// TIA Portal V17 export
// export: Created 2026-08-04T13:53:45.7641817Z, ExportSetting WithDefaults, DisplayName Totally Integrated Automation Portal, DisplayVersion V17, DisplayName TIA Portal Openness, DisplayVersion V17, DisplayName TIA Portal Version Control Interface, DisplayVersion V17, DisplayName SINAMICS Startdrive Advanced, DisplayVersion V17, DisplayName SINAMICS Startdrive G130, G150, S120, S150, SINAMICS MV, G220, S200, S210, DisplayVersion V17, DisplayName SINAMICS Startdrive G110M, G120, G120C, G120D, G120P, G115D, DisplayVersion V17, DisplayName STEP 7 Professional, DisplayVersion V17, DisplayName STEP 7 Safety, DisplayVersion V17, DisplayName WinCC Basic/Comfort/Advanced, DisplayVersion V17, DisplayName WinCC Unified, DisplayVersion V17
FUNCTION_BLOCK "Faults_FB"   // FB2, LAD
TITLE = Fault Detection
{ S7_Optimized_Access := 'TRUE' }
VERSION : 0.1
// Monitors process conditions and sets fault bits in Faults_UDT. Handles EStop detection, temperature faults, sensor health, switch conflicts, and active fault counting.
// stored: AutoNumber true, IsIECCheckEnabled false, IsRetainMemResEnabled false, MemoryReserve 100, SetENOAutomatically false, UDAEnableTagReadback false
   VAR
      Clear_Faults : "Faults_UDT";
      ons1 : Bool;
      highlimit : Real;
      TON : Array[0..10] of IEC_TIMER;
   END_VAR
   VAR_TEMP
      lowlimit : Real;
      faultcount : Int;
   END_VAR
   VAR_TEMP   // added for the SCL form of the ladder/FBD networks
      _w1 : Bool;
      _w2 : Bool;
   END_VAR
BEGIN

REGION Network 1: Fault Reset
   // Here we move a blank set of faults into our current active faults to reset them.
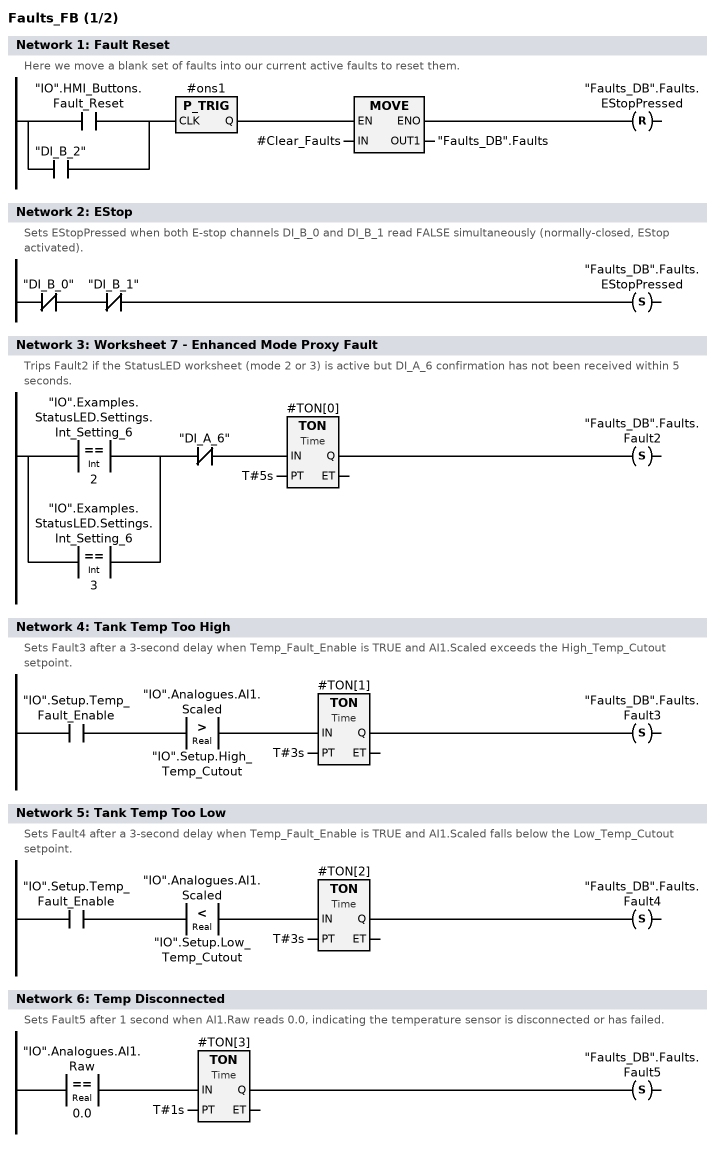
   RUNG wire#powerrail
      Contact( "IO".HMI_Buttons.Fault_Reset )
      wire#w1
      P_Trig( #ons1 )
      Move(in := #Clear_Faults, out1 => "Faults_DB".Faults)
      R_Coil( "Faults_DB".Faults.EStopPressed )
   END_RUNG
   RUNG wire#powerrail
      Contact( "DI_B_2" )
   END_RUNG wire#w1
   // the same network as SCL:
   #_w1 := "IO".HMI_Buttons.Fault_Reset OR "DI_B_2";
   #_w2 := #_w1 AND NOT #ons1;   // rising edge
   #ons1 := #_w1;
   IF #_w2 THEN
       "Faults_DB".Faults := #Clear_Faults;
       "Faults_DB".Faults.EStopPressed := FALSE;
   END_IF;
END_REGION

REGION Network 2: EStop
   // Sets EStopPressed when both E-stop channels DI_B_0 and DI_B_1 read FALSE simultaneously (normally-closed, EStop activated).
   RUNG wire#powerrail
      I_Contact( "DI_B_0" )
      I_Contact( "DI_B_1" )
      S_Coil( "Faults_DB".Faults.EStopPressed )
   END_RUNG
   // the same network as SCL:
   IF NOT "DI_B_0" AND NOT "DI_B_1" THEN "Faults_DB".Faults.EStopPressed := TRUE; END_IF;
END_REGION

REGION Network 3: Worksheet 7 - Enhanced Mode Proxy Fault
   // Trips Fault2 if the StatusLED worksheet (mode 2 or 3) is active but DI_A_6 confirmation has not been received within 5 seconds.
   RUNG wire#powerrail
      { S7_Templates := "SrcType := Int" } EQ_Contact(in1 := "IO".Examples.StatusLED.Settings.Int_Setting_6, in2 := 2)
      wire#w1
      I_Contact( "DI_A_6" )
      { S7_Templates := "time_type := Time" } #TON[0].TON(pt := T#5s, et =>)
      S_Coil( "Faults_DB".Faults.Fault2 )
   END_RUNG
   RUNG wire#powerrail
      { S7_Templates := "SrcType := Int" } EQ_Contact(in1 := "IO".Examples.StatusLED.Settings.Int_Setting_6, in2 := 3)
   END_RUNG wire#w1
   // the same network as SCL:
   #TON[0].TON(IN := (("IO".Examples.StatusLED.Settings.Int_Setting_6 = 2) OR ("IO".Examples.StatusLED.Settings.Int_Setting_6 = 3)) AND NOT "DI_A_6",
               PT := T#5s);
   IF #TON[0].Q THEN "Faults_DB".Faults.Fault2 := TRUE; END_IF;
END_REGION

REGION Network 4: Tank Temp Too High
   // Sets Fault3 after a 3-second delay when Temp_Fault_Enable is TRUE and AI1.Scaled exceeds the High_Temp_Cutout setpoint.
   RUNG wire#powerrail
      Contact( "IO".Setup.Temp_Fault_Enable )
      { S7_Templates := "SrcType := Real" } GT_Contact(in1 := "IO".Analogues.AI1.Scaled, in2 := "IO".Setup.High_Temp_Cutout)
      { S7_Templates := "time_type := Time" } #TON[1].TON(pt := T#3s, et =>)
      S_Coil( "Faults_DB".Faults.Fault3 )
   END_RUNG
   // the same network as SCL:
   #TON[1].TON(IN := "IO".Setup.Temp_Fault_Enable AND ("IO".Analogues.AI1.Scaled > "IO".Setup.High_Temp_Cutout),
               PT := T#3s);
   IF #TON[1].Q THEN "Faults_DB".Faults.Fault3 := TRUE; END_IF;
END_REGION

REGION Network 5: Tank Temp Too Low
   // Sets Fault4 after a 3-second delay when Temp_Fault_Enable is TRUE and AI1.Scaled falls below the Low_Temp_Cutout setpoint.
   RUNG wire#powerrail
      Contact( "IO".Setup.Temp_Fault_Enable )
      { S7_Templates := "SrcType := Real" } LT_Contact(in1 := "IO".Analogues.AI1.Scaled, in2 := "IO".Setup.Low_Temp_Cutout)
      { S7_Templates := "time_type := Time" } #TON[2].TON(pt := T#3s, et =>)
      S_Coil( "Faults_DB".Faults.Fault4 )
   END_RUNG
   // the same network as SCL:
   #TON[2].TON(IN := "IO".Setup.Temp_Fault_Enable AND ("IO".Analogues.AI1.Scaled < "IO".Setup.Low_Temp_Cutout),
               PT := T#3s);
   IF #TON[2].Q THEN "Faults_DB".Faults.Fault4 := TRUE; END_IF;
END_REGION

REGION Network 6: Temp Disconnected
   // Sets Fault5 after 1 second when AI1.Raw reads 0.0, indicating the temperature sensor is disconnected or has failed.
   RUNG wire#powerrail
      { S7_Templates := "SrcType := Real" } EQ_Contact(in1 := "IO".Analogues.AI1.Raw, in2 := 0.0)
      { S7_Templates := "time_type := Time" } #TON[3].TON(pt := T#1s, et =>)
      S_Coil( "Faults_DB".Faults.Fault5 )
   END_RUNG
   // the same network as SCL:
   #TON[3].TON(IN := "IO".Analogues.AI1.Raw = 0.0, PT := T#1s);
   IF #TON[3].Q THEN "Faults_DB".Faults.Fault5 := TRUE; END_IF;
END_REGION

REGION Network 7: AI0 Out of Bounds
   // Sets Fault6 after 1 second when AI0.Raw is outside the valid 0-28000 range, indicating a potentiometer fault or wiring issue.
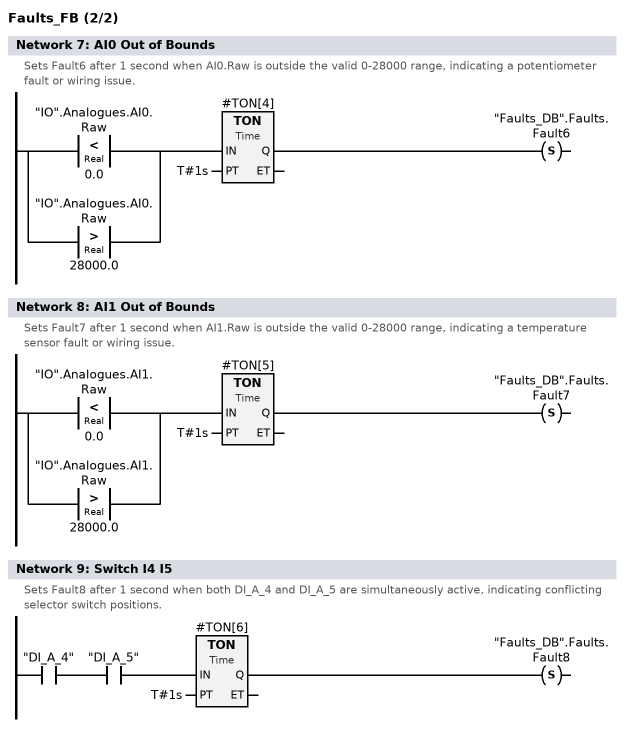
   RUNG wire#powerrail
      { S7_Templates := "SrcType := Real" } LT_Contact(in1 := "IO".Analogues.AI0.Raw, in2 := 0.0)
      wire#w1
      { S7_Templates := "time_type := Time" } #TON[4].TON(pt := T#1s, et =>)
      S_Coil( "Faults_DB".Faults.Fault6 )
   END_RUNG
   RUNG wire#powerrail
      { S7_Templates := "SrcType := Real" } GT_Contact(in1 := "IO".Analogues.AI0.Raw, in2 := 28000.0)
   END_RUNG wire#w1
   // the same network as SCL:
   #TON[4].TON(IN := ("IO".Analogues.AI0.Raw < 0.0) OR ("IO".Analogues.AI0.Raw > 28000.0), PT := T#1s);
   IF #TON[4].Q THEN "Faults_DB".Faults.Fault6 := TRUE; END_IF;
END_REGION

REGION Network 8: AI1 Out of Bounds
   // Sets Fault7 after 1 second when AI1.Raw is outside the valid 0-28000 range, indicating a temperature sensor fault or wiring issue.
   RUNG wire#powerrail
      { S7_Templates := "SrcType := Real" } LT_Contact(in1 := "IO".Analogues.AI1.Raw, in2 := 0.0)
      wire#w1
      { S7_Templates := "time_type := Time" } #TON[5].TON(pt := T#1s, et =>)
      S_Coil( "Faults_DB".Faults.Fault7 )
   END_RUNG
   RUNG wire#powerrail
      { S7_Templates := "SrcType := Real" } GT_Contact(in1 := "IO".Analogues.AI1.Raw, in2 := 28000.0)
   END_RUNG wire#w1
   // the same network as SCL:
   #TON[5].TON(IN := ("IO".Analogues.AI1.Raw < 0.0) OR ("IO".Analogues.AI1.Raw > 28000.0), PT := T#1s);
   IF #TON[5].Q THEN "Faults_DB".Faults.Fault7 := TRUE; END_IF;
END_REGION

REGION Network 9: Switch I4 I5
   // Sets Fault8 after 1 second when both DI_A_4 and DI_A_5 are simultaneously active, indicating conflicting selector switch positions.
   RUNG wire#powerrail
      Contact( "DI_A_4" )
      Contact( "DI_A_5" )
      { S7_Templates := "time_type := Time" } #TON[6].TON(pt := T#1s, et =>)
      S_Coil( "Faults_DB".Faults.Fault8 )
   END_RUNG
   // the same network as SCL:
   #TON[6].TON(IN := "DI_A_4" AND "DI_A_5", PT := T#1s);
   IF #TON[6].Q THEN "Faults_DB".Faults.Fault8 := TRUE; END_IF;
END_REGION

REGION Network 10 (SCL): Fault Count
   // Counts all active fault bits (EStopPressed plus Fault2 through Fault14) and writes the running total to Faults_DB.Faults_Count.
   // Reset the fault count to 0
   #faultcount := 0;

   // Check each fault in the Faults_UDT structure and increment the count if the fault is active
   IF "Faults_DB".Faults.EStopPressed THEN
       #faultcount := #faultcount + 1;
   END_IF;

   IF "Faults_DB".Faults.Fault2 THEN
       #faultcount := #faultcount + 1;
   END_IF;

   IF "Faults_DB".Faults.Fault3 THEN
       #faultcount := #faultcount + 1;
   END_IF;

   IF "Faults_DB".Faults.Fault4 THEN
       #faultcount := #faultcount + 1;
   END_IF;

   IF "Faults_DB".Faults.Fault5 THEN
       #faultcount := #faultcount + 1;
   END_IF;

   IF "Faults_DB".Faults.Fault6 THEN
       #faultcount := #faultcount + 1;
   END_IF;

   IF "Faults_DB".Faults.Fault7 THEN
       #faultcount := #faultcount + 1;
   END_IF;

   IF "Faults_DB".Faults.Fault8 THEN
       #faultcount := #faultcount + 1;
   END_IF;

   IF "Faults_DB".Faults.Fault9 THEN
       #faultcount := #faultcount + 1;
   END_IF;

   IF "Faults_DB".Faults.Fault10 THEN
       #faultcount := #faultcount + 1;
   END_IF;

   IF "Faults_DB".Faults.Fault11 THEN
       #faultcount := #faultcount + 1;
   END_IF;

   IF "Faults_DB".Faults.Fault12 THEN
       #faultcount := #faultcount + 1;
   END_IF;

   IF "Faults_DB".Faults.Fault13 THEN
       #faultcount := #faultcount + 1;
   END_IF;

   IF "Faults_DB".Faults.Fault14 THEN
       #faultcount := #faultcount + 1;
   END_IF;

   "Faults_DB".Faults_Count := #faultcount;
END_REGION
END_FUNCTION_BLOCK
